// TIA Portal V18 export
FUNCTION "_buttonsAndLEDs_main" : Void   // FC6, FBD
{ S7_Optimized_Access := 'TRUE' }
VERSION : 0.1
// stored: AutoNumber true, IsIECCheckEnabled false, SetENOAutomatically false, UDAEnableTagReadback false
BEGIN

REGION Network 1
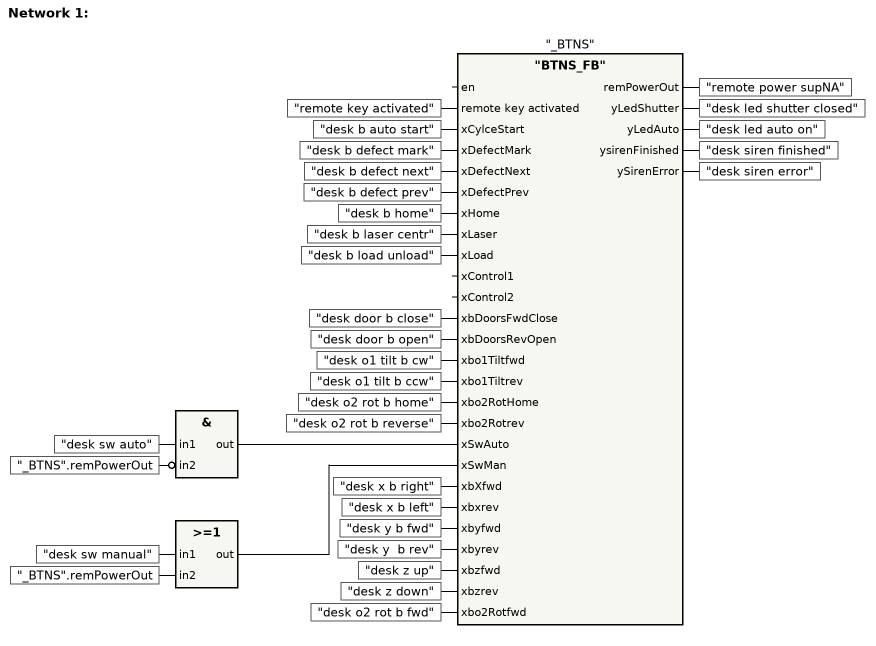
   "_BTNS"("remote key activated" := "remote key activated",   // "BTNS_FB"
           xCylceStart := "desk b auto start",
           xDefectMark := "desk b defect mark",
           xDefectNext := "desk b defect next",
           xDefectPrev := "desk b defect prev",
           xHome := "desk b home",
           xLaser := "desk b laser centr",
           xLoad := "desk b load unload",
           xbDoorsFwdClose := "desk door b close",
           xbDoorsRevOpen := "desk door b open",
           xbo1Tiltfwd := "desk o1 tilt b cw",
           xbo1Tiltrev := "desk o1 tilt b ccw",
           xbo2RotHome := "desk o2 rot b home",
           xbo2Rotrev := "desk o2 rot b reverse",
           xSwAuto := "desk sw auto" AND NOT "_BTNS".remPowerOut,
           xSwMan := "desk sw manual" OR "_BTNS".remPowerOut,
           xbXfwd := "desk x b right",
           xbxrev := "desk x b left",
           xbyfwd := "desk y b fwd",
           xbyrev := "desk y  b rev",
           xbzfwd := "desk z up",
           xbzrev := "desk z down",
           xbo2Rotfwd := "desk o2 rot b fwd",
           remPowerOut => "remote power supNA",
           yLedShutter => "desk led shutter closed",
           yLedAuto => "desk led auto on",
           ysirenFinished => "desk siren finished",
           ySirenError => "desk siren error");
END_REGION
END_FUNCTION
